// TIA Portal V18 export
FUNCTION "SS1_A1_CPU1215_IO_Update" : Void   // FC11010, LAD
{ S7_Optimized_Access := 'TRUE' }
VERSION : 0.1
// stored: AutoNumber false, IsIECCheckEnabled false, SetENOAutomatically false, UDAEnableTagReadback false
BEGIN

REGION Network 1: AI0 / "AI01.1.1" iw64
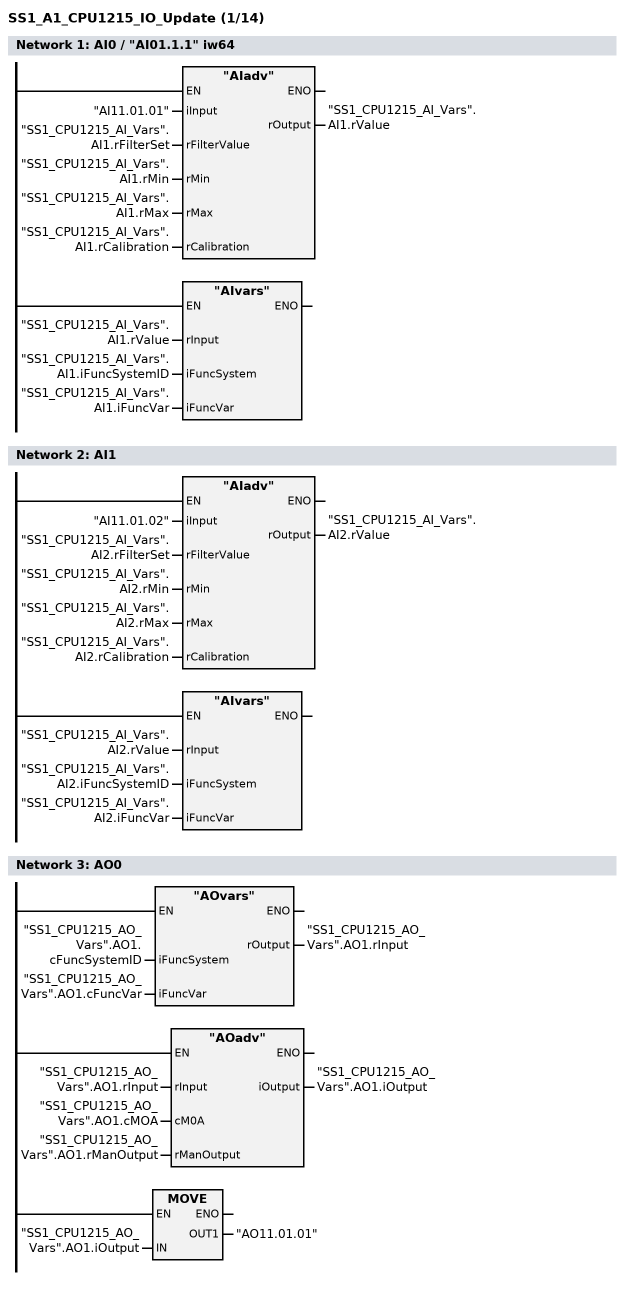
   RUNG wire#powerrail
      "AIadv"(iInput := "AI11.01.01", rFilterValue := "SS1_CPU1215_AI_Vars".AI1.rFilterSet, rMin := "SS1_CPU1215_AI_Vars".AI1.rMin, rMax := "SS1_CPU1215_AI_Vars".AI1.rMax, rCalibration := "SS1_CPU1215_AI_Vars".AI1.rCalibration, rOutput => "SS1_CPU1215_AI_Vars".AI1.rValue)
   END_RUNG
   RUNG wire#powerrail
      "AIvars"(rInput := "SS1_CPU1215_AI_Vars".AI1.rValue, iFuncSystem := "SS1_CPU1215_AI_Vars".AI1.iFuncSystemID, iFuncVar := "SS1_CPU1215_AI_Vars".AI1.iFuncVar)
   END_RUNG
   // the same network as SCL:
   "AIadv"(iInput := "AI11.01.01",
           rFilterValue := "SS1_CPU1215_AI_Vars".AI1.rFilterSet,
           rMin := "SS1_CPU1215_AI_Vars".AI1.rMin,
           rMax := "SS1_CPU1215_AI_Vars".AI1.rMax,
           rCalibration := "SS1_CPU1215_AI_Vars".AI1.rCalibration,
           rOutput => "SS1_CPU1215_AI_Vars".AI1.rValue);
   "AIvars"(rInput := "SS1_CPU1215_AI_Vars".AI1.rValue,
            iFuncSystem := "SS1_CPU1215_AI_Vars".AI1.iFuncSystemID,
            iFuncVar := "SS1_CPU1215_AI_Vars".AI1.iFuncVar);
END_REGION

REGION Network 2: AI1
   RUNG wire#powerrail
      "AIadv"(iInput := "AI11.01.02", rFilterValue := "SS1_CPU1215_AI_Vars".AI2.rFilterSet, rMin := "SS1_CPU1215_AI_Vars".AI2.rMin, rMax := "SS1_CPU1215_AI_Vars".AI2.rMax, rCalibration := "SS1_CPU1215_AI_Vars".AI2.rCalibration, rOutput => "SS1_CPU1215_AI_Vars".AI2.rValue)
   END_RUNG
   RUNG wire#powerrail
      "AIvars"(rInput := "SS1_CPU1215_AI_Vars".AI2.rValue, iFuncSystem := "SS1_CPU1215_AI_Vars".AI2.iFuncSystemID, iFuncVar := "SS1_CPU1215_AI_Vars".AI2.iFuncVar)
   END_RUNG
   // the same network as SCL:
   "AIadv"(iInput := "AI11.01.02",
           rFilterValue := "SS1_CPU1215_AI_Vars".AI2.rFilterSet,
           rMin := "SS1_CPU1215_AI_Vars".AI2.rMin,
           rMax := "SS1_CPU1215_AI_Vars".AI2.rMax,
           rCalibration := "SS1_CPU1215_AI_Vars".AI2.rCalibration,
           rOutput => "SS1_CPU1215_AI_Vars".AI2.rValue);
   "AIvars"(rInput := "SS1_CPU1215_AI_Vars".AI2.rValue,
            iFuncSystem := "SS1_CPU1215_AI_Vars".AI2.iFuncSystemID,
            iFuncVar := "SS1_CPU1215_AI_Vars".AI2.iFuncVar);
END_REGION

REGION Network 3: AO0
   RUNG wire#powerrail
      "AOvars"(iFuncSystem := "SS1_CPU1215_AO_Vars".AO1.cFuncSystemID, iFuncVar := "SS1_CPU1215_AO_Vars".AO1.cFuncVar, rOutput => "SS1_CPU1215_AO_Vars".AO1.rInput)
   END_RUNG
   RUNG wire#powerrail
      "AOadv"(rInput := "SS1_CPU1215_AO_Vars".AO1.rInput, cM0A := "SS1_CPU1215_AO_Vars".AO1.cMOA, rManOutput := "SS1_CPU1215_AO_Vars".AO1.rManOutput, iOutput => "SS1_CPU1215_AO_Vars".AO1.iOutput)
   END_RUNG
   RUNG wire#powerrail
      Move(in := "SS1_CPU1215_AO_Vars".AO1.iOutput, out1 => "AO11.01.01")
   END_RUNG
   // the same network as SCL:
   "AOvars"(iFuncSystem := "SS1_CPU1215_AO_Vars".AO1.cFuncSystemID,
            iFuncVar := "SS1_CPU1215_AO_Vars".AO1.cFuncVar,
            rOutput => "SS1_CPU1215_AO_Vars".AO1.rInput);
   "AOadv"(rInput := "SS1_CPU1215_AO_Vars".AO1.rInput,
           cM0A := "SS1_CPU1215_AO_Vars".AO1.cMOA,
           rManOutput := "SS1_CPU1215_AO_Vars".AO1.rManOutput,
           iOutput => "SS1_CPU1215_AO_Vars".AO1.iOutput);
   "AO11.01.01" := "SS1_CPU1215_AO_Vars".AO1.iOutput;
END_REGION

REGION Network 4: AO1
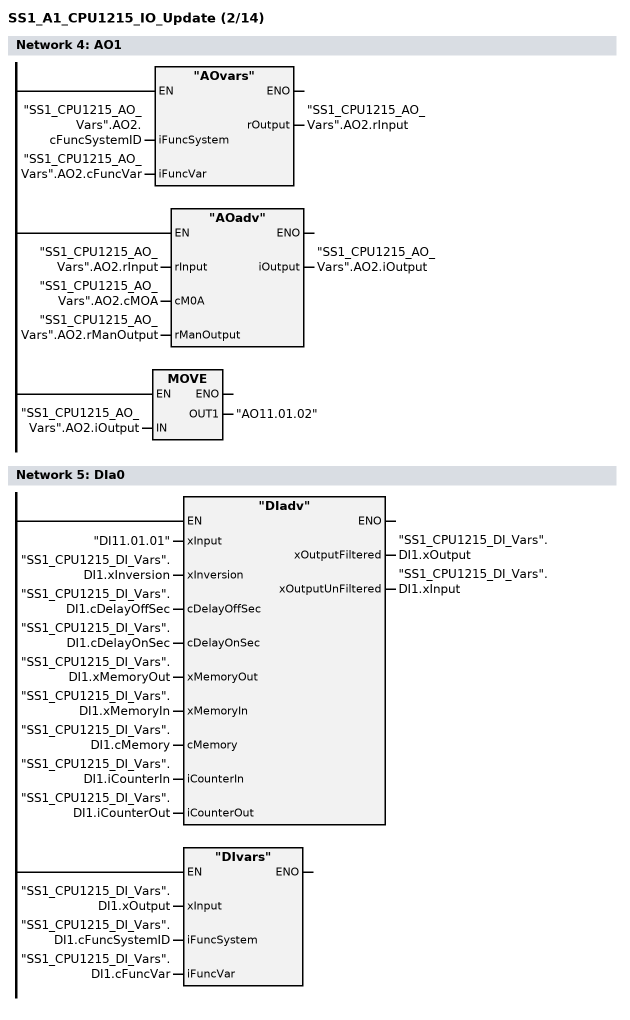
   RUNG wire#powerrail
      "AOvars"(iFuncSystem := "SS1_CPU1215_AO_Vars".AO2.cFuncSystemID, iFuncVar := "SS1_CPU1215_AO_Vars".AO2.cFuncVar, rOutput => "SS1_CPU1215_AO_Vars".AO2.rInput)
   END_RUNG
   RUNG wire#powerrail
      "AOadv"(rInput := "SS1_CPU1215_AO_Vars".AO2.rInput, cM0A := "SS1_CPU1215_AO_Vars".AO2.cMOA, rManOutput := "SS1_CPU1215_AO_Vars".AO2.rManOutput, iOutput => "SS1_CPU1215_AO_Vars".AO2.iOutput)
   END_RUNG
   RUNG wire#powerrail
      Move(in := "SS1_CPU1215_AO_Vars".AO2.iOutput, out1 => "AO11.01.02")
   END_RUNG
   // the same network as SCL:
   "AOvars"(iFuncSystem := "SS1_CPU1215_AO_Vars".AO2.cFuncSystemID,
            iFuncVar := "SS1_CPU1215_AO_Vars".AO2.cFuncVar,
            rOutput => "SS1_CPU1215_AO_Vars".AO2.rInput);
   "AOadv"(rInput := "SS1_CPU1215_AO_Vars".AO2.rInput,
           cM0A := "SS1_CPU1215_AO_Vars".AO2.cMOA,
           rManOutput := "SS1_CPU1215_AO_Vars".AO2.rManOutput,
           iOutput => "SS1_CPU1215_AO_Vars".AO2.iOutput);
   "AO11.01.02" := "SS1_CPU1215_AO_Vars".AO2.iOutput;
END_REGION

REGION Network 5: DIa0
   RUNG wire#powerrail
      "DIadv"(xInput := "DI11.01.01", xInversion := "SS1_CPU1215_DI_Vars".DI1.xInversion, cDelayOffSec := "SS1_CPU1215_DI_Vars".DI1.cDelayOffSec, cDelayOnSec := "SS1_CPU1215_DI_Vars".DI1.cDelayOnSec, xMemoryOut := "SS1_CPU1215_DI_Vars".DI1.xMemoryOut, xMemoryIn := "SS1_CPU1215_DI_Vars".DI1.xMemoryIn, cMemory := "SS1_CPU1215_DI_Vars".DI1.cMemory, xOutputFiltered => "SS1_CPU1215_DI_Vars".DI1.xOutput, xOutputUnFiltered => "SS1_CPU1215_DI_Vars".DI1.xInput, iCounterIn := "SS1_CPU1215_DI_Vars".DI1.iCounterIn, iCounterOut := "SS1_CPU1215_DI_Vars".DI1.iCounterOut)
   END_RUNG
   RUNG wire#powerrail
      "DIvars"(xInput := "SS1_CPU1215_DI_Vars".DI1.xOutput, iFuncSystem := "SS1_CPU1215_DI_Vars".DI1.cFuncSystemID, iFuncVar := "SS1_CPU1215_DI_Vars".DI1.cFuncVar)
   END_RUNG
   // the same network as SCL:
   "DIadv"(xInput := "DI11.01.01",
           xInversion := "SS1_CPU1215_DI_Vars".DI1.xInversion,
           cDelayOffSec := "SS1_CPU1215_DI_Vars".DI1.cDelayOffSec,
           cDelayOnSec := "SS1_CPU1215_DI_Vars".DI1.cDelayOnSec,
           xMemoryOut := "SS1_CPU1215_DI_Vars".DI1.xMemoryOut,
           xMemoryIn := "SS1_CPU1215_DI_Vars".DI1.xMemoryIn,
           cMemory := "SS1_CPU1215_DI_Vars".DI1.cMemory,
           iCounterIn := "SS1_CPU1215_DI_Vars".DI1.iCounterIn,
           iCounterOut := "SS1_CPU1215_DI_Vars".DI1.iCounterOut,
           xOutputFiltered => "SS1_CPU1215_DI_Vars".DI1.xOutput,
           xOutputUnFiltered => "SS1_CPU1215_DI_Vars".DI1.xInput);
   "DIvars"(xInput := "SS1_CPU1215_DI_Vars".DI1.xOutput,
            iFuncSystem := "SS1_CPU1215_DI_Vars".DI1.cFuncSystemID,
            iFuncVar := "SS1_CPU1215_DI_Vars".DI1.cFuncVar);
END_REGION

REGION Network 6: DIa1
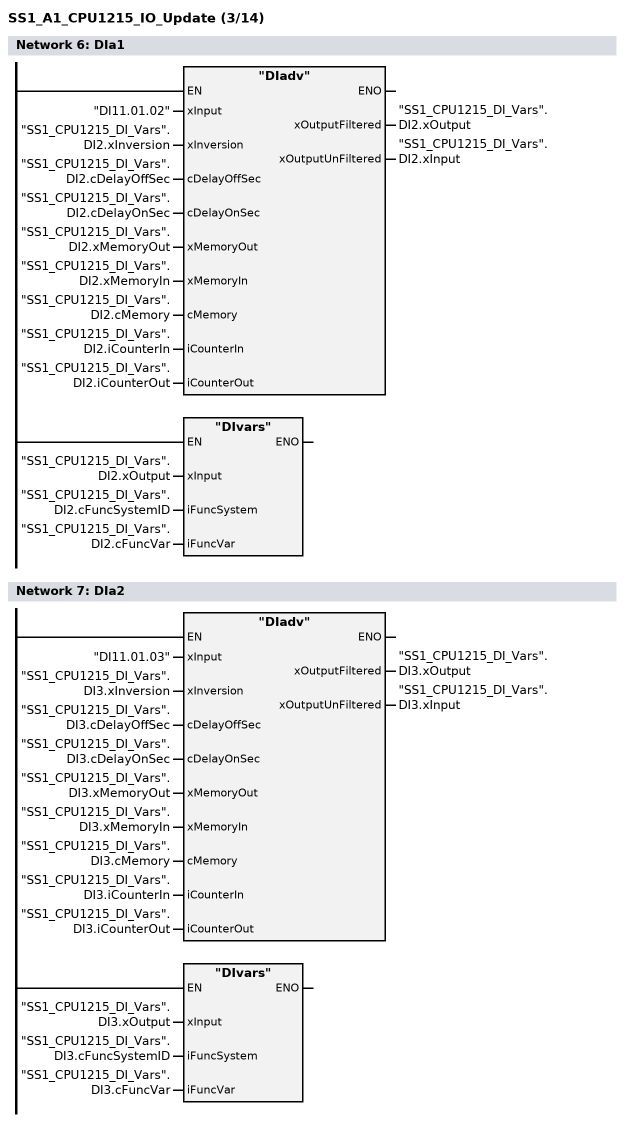
   RUNG wire#powerrail
      "DIadv"(xInput := "DI11.01.02", xInversion := "SS1_CPU1215_DI_Vars".DI2.xInversion, cDelayOffSec := "SS1_CPU1215_DI_Vars".DI2.cDelayOffSec, cDelayOnSec := "SS1_CPU1215_DI_Vars".DI2.cDelayOnSec, xMemoryOut := "SS1_CPU1215_DI_Vars".DI2.xMemoryOut, xMemoryIn := "SS1_CPU1215_DI_Vars".DI2.xMemoryIn, cMemory := "SS1_CPU1215_DI_Vars".DI2.cMemory, xOutputFiltered => "SS1_CPU1215_DI_Vars".DI2.xOutput, xOutputUnFiltered => "SS1_CPU1215_DI_Vars".DI2.xInput, iCounterIn := "SS1_CPU1215_DI_Vars".DI2.iCounterIn, iCounterOut := "SS1_CPU1215_DI_Vars".DI2.iCounterOut)
   END_RUNG
   RUNG wire#powerrail
      "DIvars"(xInput := "SS1_CPU1215_DI_Vars".DI2.xOutput, iFuncSystem := "SS1_CPU1215_DI_Vars".DI2.cFuncSystemID, iFuncVar := "SS1_CPU1215_DI_Vars".DI2.cFuncVar)
   END_RUNG
   // the same network as SCL:
   "DIadv"(xInput := "DI11.01.02",
           xInversion := "SS1_CPU1215_DI_Vars".DI2.xInversion,
           cDelayOffSec := "SS1_CPU1215_DI_Vars".DI2.cDelayOffSec,
           cDelayOnSec := "SS1_CPU1215_DI_Vars".DI2.cDelayOnSec,
           xMemoryOut := "SS1_CPU1215_DI_Vars".DI2.xMemoryOut,
           xMemoryIn := "SS1_CPU1215_DI_Vars".DI2.xMemoryIn,
           cMemory := "SS1_CPU1215_DI_Vars".DI2.cMemory,
           iCounterIn := "SS1_CPU1215_DI_Vars".DI2.iCounterIn,
           iCounterOut := "SS1_CPU1215_DI_Vars".DI2.iCounterOut,
           xOutputFiltered => "SS1_CPU1215_DI_Vars".DI2.xOutput,
           xOutputUnFiltered => "SS1_CPU1215_DI_Vars".DI2.xInput);
   "DIvars"(xInput := "SS1_CPU1215_DI_Vars".DI2.xOutput,
            iFuncSystem := "SS1_CPU1215_DI_Vars".DI2.cFuncSystemID,
            iFuncVar := "SS1_CPU1215_DI_Vars".DI2.cFuncVar);
END_REGION

REGION Network 7: DIa2
   RUNG wire#powerrail
      "DIadv"(xInput := "DI11.01.03", xInversion := "SS1_CPU1215_DI_Vars".DI3.xInversion, cDelayOffSec := "SS1_CPU1215_DI_Vars".DI3.cDelayOffSec, cDelayOnSec := "SS1_CPU1215_DI_Vars".DI3.cDelayOnSec, xMemoryOut := "SS1_CPU1215_DI_Vars".DI3.xMemoryOut, xMemoryIn := "SS1_CPU1215_DI_Vars".DI3.xMemoryIn, cMemory := "SS1_CPU1215_DI_Vars".DI3.cMemory, xOutputFiltered => "SS1_CPU1215_DI_Vars".DI3.xOutput, xOutputUnFiltered => "SS1_CPU1215_DI_Vars".DI3.xInput, iCounterIn := "SS1_CPU1215_DI_Vars".DI3.iCounterIn, iCounterOut := "SS1_CPU1215_DI_Vars".DI3.iCounterOut)
   END_RUNG
   RUNG wire#powerrail
      "DIvars"(xInput := "SS1_CPU1215_DI_Vars".DI3.xOutput, iFuncSystem := "SS1_CPU1215_DI_Vars".DI3.cFuncSystemID, iFuncVar := "SS1_CPU1215_DI_Vars".DI3.cFuncVar)
   END_RUNG
   // the same network as SCL:
   "DIadv"(xInput := "DI11.01.03",
           xInversion := "SS1_CPU1215_DI_Vars".DI3.xInversion,
           cDelayOffSec := "SS1_CPU1215_DI_Vars".DI3.cDelayOffSec,
           cDelayOnSec := "SS1_CPU1215_DI_Vars".DI3.cDelayOnSec,
           xMemoryOut := "SS1_CPU1215_DI_Vars".DI3.xMemoryOut,
           xMemoryIn := "SS1_CPU1215_DI_Vars".DI3.xMemoryIn,
           cMemory := "SS1_CPU1215_DI_Vars".DI3.cMemory,
           iCounterIn := "SS1_CPU1215_DI_Vars".DI3.iCounterIn,
           iCounterOut := "SS1_CPU1215_DI_Vars".DI3.iCounterOut,
           xOutputFiltered => "SS1_CPU1215_DI_Vars".DI3.xOutput,
           xOutputUnFiltered => "SS1_CPU1215_DI_Vars".DI3.xInput);
   "DIvars"(xInput := "SS1_CPU1215_DI_Vars".DI3.xOutput,
            iFuncSystem := "SS1_CPU1215_DI_Vars".DI3.cFuncSystemID,
            iFuncVar := "SS1_CPU1215_DI_Vars".DI3.cFuncVar);
END_REGION

REGION Network 8: DIa3
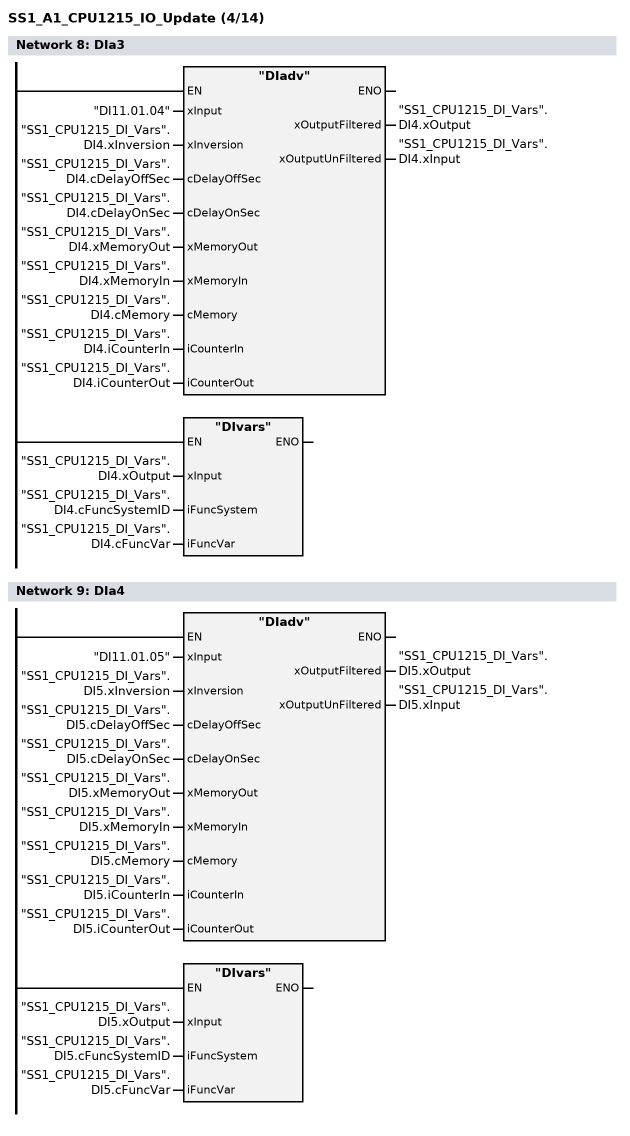
   RUNG wire#powerrail
      "DIadv"(xInput := "DI11.01.04", xInversion := "SS1_CPU1215_DI_Vars".DI4.xInversion, cDelayOffSec := "SS1_CPU1215_DI_Vars".DI4.cDelayOffSec, cDelayOnSec := "SS1_CPU1215_DI_Vars".DI4.cDelayOnSec, xMemoryOut := "SS1_CPU1215_DI_Vars".DI4.xMemoryOut, xMemoryIn := "SS1_CPU1215_DI_Vars".DI4.xMemoryIn, cMemory := "SS1_CPU1215_DI_Vars".DI4.cMemory, xOutputFiltered => "SS1_CPU1215_DI_Vars".DI4.xOutput, xOutputUnFiltered => "SS1_CPU1215_DI_Vars".DI4.xInput, iCounterIn := "SS1_CPU1215_DI_Vars".DI4.iCounterIn, iCounterOut := "SS1_CPU1215_DI_Vars".DI4.iCounterOut)
   END_RUNG
   RUNG wire#powerrail
      "DIvars"(xInput := "SS1_CPU1215_DI_Vars".DI4.xOutput, iFuncSystem := "SS1_CPU1215_DI_Vars".DI4.cFuncSystemID, iFuncVar := "SS1_CPU1215_DI_Vars".DI4.cFuncVar)
   END_RUNG
   // the same network as SCL:
   "DIadv"(xInput := "DI11.01.04",
           xInversion := "SS1_CPU1215_DI_Vars".DI4.xInversion,
           cDelayOffSec := "SS1_CPU1215_DI_Vars".DI4.cDelayOffSec,
           cDelayOnSec := "SS1_CPU1215_DI_Vars".DI4.cDelayOnSec,
           xMemoryOut := "SS1_CPU1215_DI_Vars".DI4.xMemoryOut,
           xMemoryIn := "SS1_CPU1215_DI_Vars".DI4.xMemoryIn,
           cMemory := "SS1_CPU1215_DI_Vars".DI4.cMemory,
           iCounterIn := "SS1_CPU1215_DI_Vars".DI4.iCounterIn,
           iCounterOut := "SS1_CPU1215_DI_Vars".DI4.iCounterOut,
           xOutputFiltered => "SS1_CPU1215_DI_Vars".DI4.xOutput,
           xOutputUnFiltered => "SS1_CPU1215_DI_Vars".DI4.xInput);
   "DIvars"(xInput := "SS1_CPU1215_DI_Vars".DI4.xOutput,
            iFuncSystem := "SS1_CPU1215_DI_Vars".DI4.cFuncSystemID,
            iFuncVar := "SS1_CPU1215_DI_Vars".DI4.cFuncVar);
END_REGION

REGION Network 9: DIa4
   RUNG wire#powerrail
      "DIadv"(xInput := "DI11.01.05", xInversion := "SS1_CPU1215_DI_Vars".DI5.xInversion, cDelayOffSec := "SS1_CPU1215_DI_Vars".DI5.cDelayOffSec, cDelayOnSec := "SS1_CPU1215_DI_Vars".DI5.cDelayOnSec, xMemoryOut := "SS1_CPU1215_DI_Vars".DI5.xMemoryOut, xMemoryIn := "SS1_CPU1215_DI_Vars".DI5.xMemoryIn, cMemory := "SS1_CPU1215_DI_Vars".DI5.cMemory, xOutputFiltered => "SS1_CPU1215_DI_Vars".DI5.xOutput, xOutputUnFiltered => "SS1_CPU1215_DI_Vars".DI5.xInput, iCounterIn := "SS1_CPU1215_DI_Vars".DI5.iCounterIn, iCounterOut := "SS1_CPU1215_DI_Vars".DI5.iCounterOut)
   END_RUNG
   RUNG wire#powerrail
      "DIvars"(xInput := "SS1_CPU1215_DI_Vars".DI5.xOutput, iFuncSystem := "SS1_CPU1215_DI_Vars".DI5.cFuncSystemID, iFuncVar := "SS1_CPU1215_DI_Vars".DI5.cFuncVar)
   END_RUNG
   // the same network as SCL:
   "DIadv"(xInput := "DI11.01.05",
           xInversion := "SS1_CPU1215_DI_Vars".DI5.xInversion,
           cDelayOffSec := "SS1_CPU1215_DI_Vars".DI5.cDelayOffSec,
           cDelayOnSec := "SS1_CPU1215_DI_Vars".DI5.cDelayOnSec,
           xMemoryOut := "SS1_CPU1215_DI_Vars".DI5.xMemoryOut,
           xMemoryIn := "SS1_CPU1215_DI_Vars".DI5.xMemoryIn,
           cMemory := "SS1_CPU1215_DI_Vars".DI5.cMemory,
           iCounterIn := "SS1_CPU1215_DI_Vars".DI5.iCounterIn,
           iCounterOut := "SS1_CPU1215_DI_Vars".DI5.iCounterOut,
           xOutputFiltered => "SS1_CPU1215_DI_Vars".DI5.xOutput,
           xOutputUnFiltered => "SS1_CPU1215_DI_Vars".DI5.xInput);
   "DIvars"(xInput := "SS1_CPU1215_DI_Vars".DI5.xOutput,
            iFuncSystem := "SS1_CPU1215_DI_Vars".DI5.cFuncSystemID,
            iFuncVar := "SS1_CPU1215_DI_Vars".DI5.cFuncVar);
END_REGION

REGION Network 10: DIa5
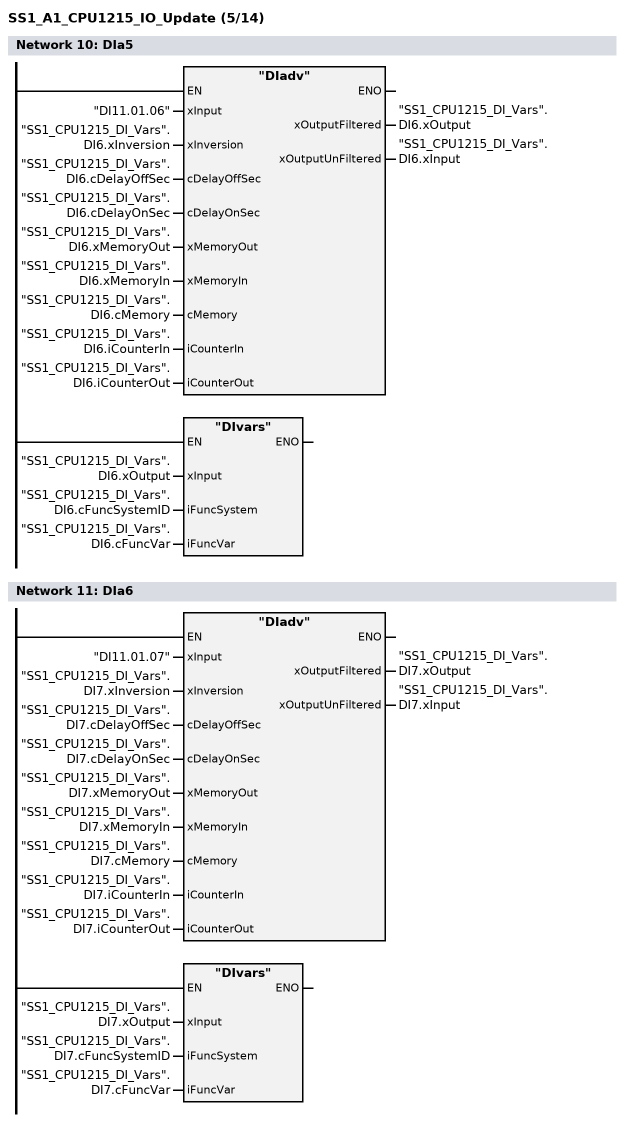
   RUNG wire#powerrail
      "DIadv"(xInput := "DI11.01.06", xInversion := "SS1_CPU1215_DI_Vars".DI6.xInversion, cDelayOffSec := "SS1_CPU1215_DI_Vars".DI6.cDelayOffSec, cDelayOnSec := "SS1_CPU1215_DI_Vars".DI6.cDelayOnSec, xMemoryOut := "SS1_CPU1215_DI_Vars".DI6.xMemoryOut, xMemoryIn := "SS1_CPU1215_DI_Vars".DI6.xMemoryIn, cMemory := "SS1_CPU1215_DI_Vars".DI6.cMemory, xOutputFiltered => "SS1_CPU1215_DI_Vars".DI6.xOutput, xOutputUnFiltered => "SS1_CPU1215_DI_Vars".DI6.xInput, iCounterIn := "SS1_CPU1215_DI_Vars".DI6.iCounterIn, iCounterOut := "SS1_CPU1215_DI_Vars".DI6.iCounterOut)
   END_RUNG
   RUNG wire#powerrail
      "DIvars"(xInput := "SS1_CPU1215_DI_Vars".DI6.xOutput, iFuncSystem := "SS1_CPU1215_DI_Vars".DI6.cFuncSystemID, iFuncVar := "SS1_CPU1215_DI_Vars".DI6.cFuncVar)
   END_RUNG
   // the same network as SCL:
   "DIadv"(xInput := "DI11.01.06",
           xInversion := "SS1_CPU1215_DI_Vars".DI6.xInversion,
           cDelayOffSec := "SS1_CPU1215_DI_Vars".DI6.cDelayOffSec,
           cDelayOnSec := "SS1_CPU1215_DI_Vars".DI6.cDelayOnSec,
           xMemoryOut := "SS1_CPU1215_DI_Vars".DI6.xMemoryOut,
           xMemoryIn := "SS1_CPU1215_DI_Vars".DI6.xMemoryIn,
           cMemory := "SS1_CPU1215_DI_Vars".DI6.cMemory,
           iCounterIn := "SS1_CPU1215_DI_Vars".DI6.iCounterIn,
           iCounterOut := "SS1_CPU1215_DI_Vars".DI6.iCounterOut,
           xOutputFiltered => "SS1_CPU1215_DI_Vars".DI6.xOutput,
           xOutputUnFiltered => "SS1_CPU1215_DI_Vars".DI6.xInput);
   "DIvars"(xInput := "SS1_CPU1215_DI_Vars".DI6.xOutput,
            iFuncSystem := "SS1_CPU1215_DI_Vars".DI6.cFuncSystemID,
            iFuncVar := "SS1_CPU1215_DI_Vars".DI6.cFuncVar);
END_REGION

REGION Network 11: DIa6
   RUNG wire#powerrail
      "DIadv"(xInput := "DI11.01.07", xInversion := "SS1_CPU1215_DI_Vars".DI7.xInversion, cDelayOffSec := "SS1_CPU1215_DI_Vars".DI7.cDelayOffSec, cDelayOnSec := "SS1_CPU1215_DI_Vars".DI7.cDelayOnSec, xMemoryOut := "SS1_CPU1215_DI_Vars".DI7.xMemoryOut, xMemoryIn := "SS1_CPU1215_DI_Vars".DI7.xMemoryIn, cMemory := "SS1_CPU1215_DI_Vars".DI7.cMemory, xOutputFiltered => "SS1_CPU1215_DI_Vars".DI7.xOutput, xOutputUnFiltered => "SS1_CPU1215_DI_Vars".DI7.xInput, iCounterIn := "SS1_CPU1215_DI_Vars".DI7.iCounterIn, iCounterOut := "SS1_CPU1215_DI_Vars".DI7.iCounterOut)
   END_RUNG
   RUNG wire#powerrail
      "DIvars"(xInput := "SS1_CPU1215_DI_Vars".DI7.xOutput, iFuncSystem := "SS1_CPU1215_DI_Vars".DI7.cFuncSystemID, iFuncVar := "SS1_CPU1215_DI_Vars".DI7.cFuncVar)
   END_RUNG
   // the same network as SCL:
   "DIadv"(xInput := "DI11.01.07",
           xInversion := "SS1_CPU1215_DI_Vars".DI7.xInversion,
           cDelayOffSec := "SS1_CPU1215_DI_Vars".DI7.cDelayOffSec,
           cDelayOnSec := "SS1_CPU1215_DI_Vars".DI7.cDelayOnSec,
           xMemoryOut := "SS1_CPU1215_DI_Vars".DI7.xMemoryOut,
           xMemoryIn := "SS1_CPU1215_DI_Vars".DI7.xMemoryIn,
           cMemory := "SS1_CPU1215_DI_Vars".DI7.cMemory,
           iCounterIn := "SS1_CPU1215_DI_Vars".DI7.iCounterIn,
           iCounterOut := "SS1_CPU1215_DI_Vars".DI7.iCounterOut,
           xOutputFiltered => "SS1_CPU1215_DI_Vars".DI7.xOutput,
           xOutputUnFiltered => "SS1_CPU1215_DI_Vars".DI7.xInput);
   "DIvars"(xInput := "SS1_CPU1215_DI_Vars".DI7.xOutput,
            iFuncSystem := "SS1_CPU1215_DI_Vars".DI7.cFuncSystemID,
            iFuncVar := "SS1_CPU1215_DI_Vars".DI7.cFuncVar);
END_REGION

REGION Network 12: DIa7 / DI01.1.08 EDP під охороною
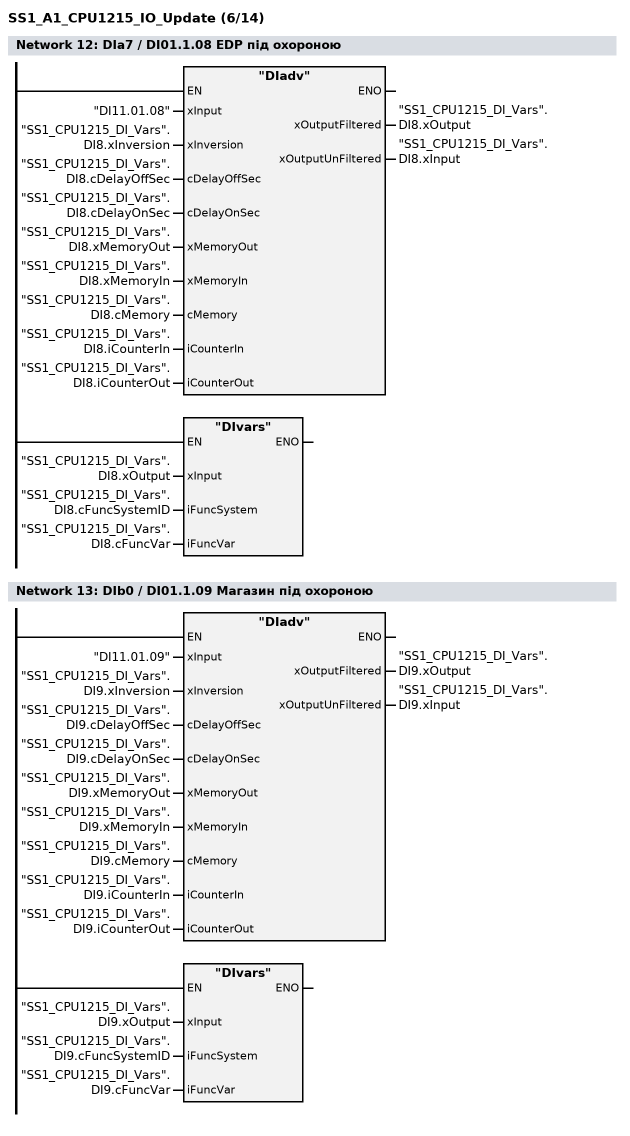
   RUNG wire#powerrail
      "DIadv"(xInput := "DI11.01.08", xInversion := "SS1_CPU1215_DI_Vars".DI8.xInversion, cDelayOffSec := "SS1_CPU1215_DI_Vars".DI8.cDelayOffSec, cDelayOnSec := "SS1_CPU1215_DI_Vars".DI8.cDelayOnSec, xMemoryOut := "SS1_CPU1215_DI_Vars".DI8.xMemoryOut, xMemoryIn := "SS1_CPU1215_DI_Vars".DI8.xMemoryIn, cMemory := "SS1_CPU1215_DI_Vars".DI8.cMemory, iCounterIn := "SS1_CPU1215_DI_Vars".DI8.iCounterIn, iCounterOut := "SS1_CPU1215_DI_Vars".DI8.iCounterOut, xOutputFiltered => "SS1_CPU1215_DI_Vars".DI8.xOutput, xOutputUnFiltered => "SS1_CPU1215_DI_Vars".DI8.xInput)
   END_RUNG
   RUNG wire#powerrail
      "DIvars"(xInput := "SS1_CPU1215_DI_Vars".DI8.xOutput, iFuncSystem := "SS1_CPU1215_DI_Vars".DI8.cFuncSystemID, iFuncVar := "SS1_CPU1215_DI_Vars".DI8.cFuncVar)
   END_RUNG
   // the same network as SCL:
   "DIadv"(xInput := "DI11.01.08",
           xInversion := "SS1_CPU1215_DI_Vars".DI8.xInversion,
           cDelayOffSec := "SS1_CPU1215_DI_Vars".DI8.cDelayOffSec,
           cDelayOnSec := "SS1_CPU1215_DI_Vars".DI8.cDelayOnSec,
           xMemoryOut := "SS1_CPU1215_DI_Vars".DI8.xMemoryOut,
           xMemoryIn := "SS1_CPU1215_DI_Vars".DI8.xMemoryIn,
           cMemory := "SS1_CPU1215_DI_Vars".DI8.cMemory,
           iCounterIn := "SS1_CPU1215_DI_Vars".DI8.iCounterIn,
           iCounterOut := "SS1_CPU1215_DI_Vars".DI8.iCounterOut,
           xOutputFiltered => "SS1_CPU1215_DI_Vars".DI8.xOutput,
           xOutputUnFiltered => "SS1_CPU1215_DI_Vars".DI8.xInput);
   "DIvars"(xInput := "SS1_CPU1215_DI_Vars".DI8.xOutput,
            iFuncSystem := "SS1_CPU1215_DI_Vars".DI8.cFuncSystemID,
            iFuncVar := "SS1_CPU1215_DI_Vars".DI8.cFuncVar);
END_REGION

REGION Network 13: DIb0 / DI01.1.09 Магазин під охороною
   RUNG wire#powerrail
      "DIadv"(xInput := "DI11.01.09", xInversion := "SS1_CPU1215_DI_Vars".DI9.xInversion, cDelayOffSec := "SS1_CPU1215_DI_Vars".DI9.cDelayOffSec, cDelayOnSec := "SS1_CPU1215_DI_Vars".DI9.cDelayOnSec, xMemoryOut := "SS1_CPU1215_DI_Vars".DI9.xMemoryOut, xMemoryIn := "SS1_CPU1215_DI_Vars".DI9.xMemoryIn, cMemory := "SS1_CPU1215_DI_Vars".DI9.cMemory, xOutputFiltered => "SS1_CPU1215_DI_Vars".DI9.xOutput, xOutputUnFiltered => "SS1_CPU1215_DI_Vars".DI9.xInput, iCounterIn := "SS1_CPU1215_DI_Vars".DI9.iCounterIn, iCounterOut := "SS1_CPU1215_DI_Vars".DI9.iCounterOut)
   END_RUNG
   RUNG wire#powerrail
      "DIvars"(xInput := "SS1_CPU1215_DI_Vars".DI9.xOutput, iFuncSystem := "SS1_CPU1215_DI_Vars".DI9.cFuncSystemID, iFuncVar := "SS1_CPU1215_DI_Vars".DI9.cFuncVar)
   END_RUNG
   // the same network as SCL:
   "DIadv"(xInput := "DI11.01.09",
           xInversion := "SS1_CPU1215_DI_Vars".DI9.xInversion,
           cDelayOffSec := "SS1_CPU1215_DI_Vars".DI9.cDelayOffSec,
           cDelayOnSec := "SS1_CPU1215_DI_Vars".DI9.cDelayOnSec,
           xMemoryOut := "SS1_CPU1215_DI_Vars".DI9.xMemoryOut,
           xMemoryIn := "SS1_CPU1215_DI_Vars".DI9.xMemoryIn,
           cMemory := "SS1_CPU1215_DI_Vars".DI9.cMemory,
           iCounterIn := "SS1_CPU1215_DI_Vars".DI9.iCounterIn,
           iCounterOut := "SS1_CPU1215_DI_Vars".DI9.iCounterOut,
           xOutputFiltered => "SS1_CPU1215_DI_Vars".DI9.xOutput,
           xOutputUnFiltered => "SS1_CPU1215_DI_Vars".DI9.xInput);
   "DIvars"(xInput := "SS1_CPU1215_DI_Vars".DI9.xOutput,
            iFuncSystem := "SS1_CPU1215_DI_Vars".DI9.cFuncSystemID,
            iFuncVar := "SS1_CPU1215_DI_Vars".DI9.cFuncVar);
END_REGION

REGION Network 14: DIb1 / DI01.1.10 Аварійний рівень загазованості
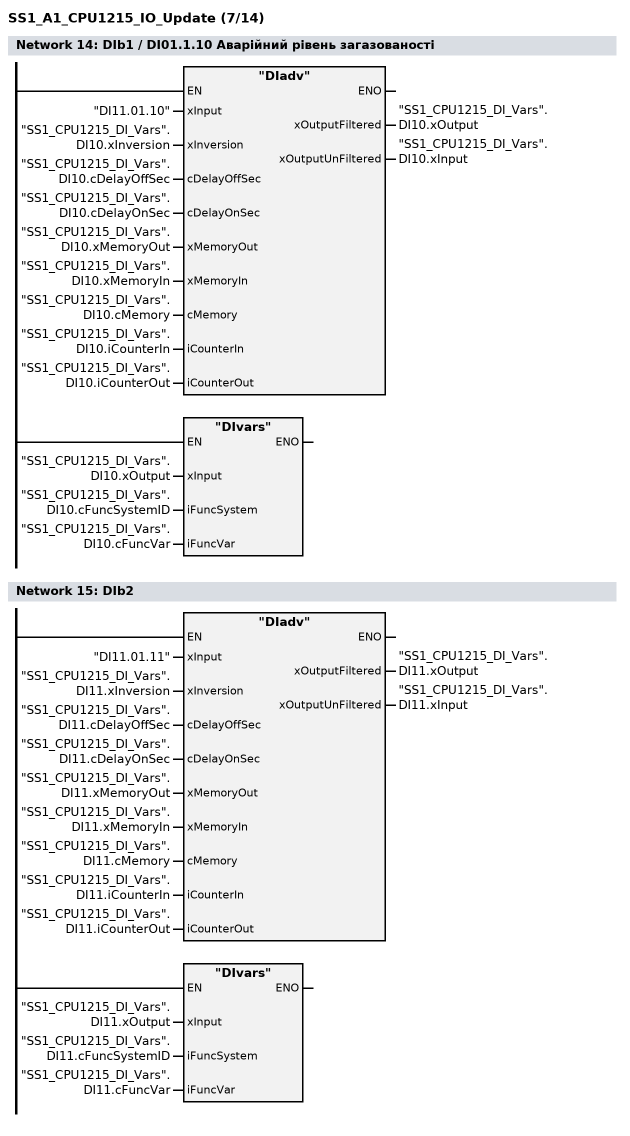
   RUNG wire#powerrail
      "DIadv"(xInput := "DI11.01.10", xInversion := "SS1_CPU1215_DI_Vars".DI10.xInversion, cDelayOffSec := "SS1_CPU1215_DI_Vars".DI10.cDelayOffSec, cDelayOnSec := "SS1_CPU1215_DI_Vars".DI10.cDelayOnSec, xMemoryOut := "SS1_CPU1215_DI_Vars".DI10.xMemoryOut, xMemoryIn := "SS1_CPU1215_DI_Vars".DI10.xMemoryIn, cMemory := "SS1_CPU1215_DI_Vars".DI10.cMemory, xOutputFiltered => "SS1_CPU1215_DI_Vars".DI10.xOutput, xOutputUnFiltered => "SS1_CPU1215_DI_Vars".DI10.xInput, iCounterIn := "SS1_CPU1215_DI_Vars".DI10.iCounterIn, iCounterOut := "SS1_CPU1215_DI_Vars".DI10.iCounterOut)
   END_RUNG
   RUNG wire#powerrail
      "DIvars"(xInput := "SS1_CPU1215_DI_Vars".DI10.xOutput, iFuncSystem := "SS1_CPU1215_DI_Vars".DI10.cFuncSystemID, iFuncVar := "SS1_CPU1215_DI_Vars".DI10.cFuncVar)
   END_RUNG
   // the same network as SCL:
   "DIadv"(xInput := "DI11.01.10",
           xInversion := "SS1_CPU1215_DI_Vars".DI10.xInversion,
           cDelayOffSec := "SS1_CPU1215_DI_Vars".DI10.cDelayOffSec,
           cDelayOnSec := "SS1_CPU1215_DI_Vars".DI10.cDelayOnSec,
           xMemoryOut := "SS1_CPU1215_DI_Vars".DI10.xMemoryOut,
           xMemoryIn := "SS1_CPU1215_DI_Vars".DI10.xMemoryIn,
           cMemory := "SS1_CPU1215_DI_Vars".DI10.cMemory,
           iCounterIn := "SS1_CPU1215_DI_Vars".DI10.iCounterIn,
           iCounterOut := "SS1_CPU1215_DI_Vars".DI10.iCounterOut,
           xOutputFiltered => "SS1_CPU1215_DI_Vars".DI10.xOutput,
           xOutputUnFiltered => "SS1_CPU1215_DI_Vars".DI10.xInput);
   "DIvars"(xInput := "SS1_CPU1215_DI_Vars".DI10.xOutput,
            iFuncSystem := "SS1_CPU1215_DI_Vars".DI10.cFuncSystemID,
            iFuncVar := "SS1_CPU1215_DI_Vars".DI10.cFuncVar);
END_REGION

REGION Network 15: DIb2
   RUNG wire#powerrail
      "DIadv"(xInput := "DI11.01.11", xInversion := "SS1_CPU1215_DI_Vars".DI11.xInversion, cDelayOffSec := "SS1_CPU1215_DI_Vars".DI11.cDelayOffSec, cDelayOnSec := "SS1_CPU1215_DI_Vars".DI11.cDelayOnSec, xMemoryOut := "SS1_CPU1215_DI_Vars".DI11.xMemoryOut, xMemoryIn := "SS1_CPU1215_DI_Vars".DI11.xMemoryIn, cMemory := "SS1_CPU1215_DI_Vars".DI11.cMemory, iCounterIn := "SS1_CPU1215_DI_Vars".DI11.iCounterIn, iCounterOut := "SS1_CPU1215_DI_Vars".DI11.iCounterOut, xOutputFiltered => "SS1_CPU1215_DI_Vars".DI11.xOutput, xOutputUnFiltered => "SS1_CPU1215_DI_Vars".DI11.xInput)
   END_RUNG
   RUNG wire#powerrail
      "DIvars"(xInput := "SS1_CPU1215_DI_Vars".DI11.xOutput, iFuncSystem := "SS1_CPU1215_DI_Vars".DI11.cFuncSystemID, iFuncVar := "SS1_CPU1215_DI_Vars".DI11.cFuncVar)
   END_RUNG
   // the same network as SCL:
   "DIadv"(xInput := "DI11.01.11",
           xInversion := "SS1_CPU1215_DI_Vars".DI11.xInversion,
           cDelayOffSec := "SS1_CPU1215_DI_Vars".DI11.cDelayOffSec,
           cDelayOnSec := "SS1_CPU1215_DI_Vars".DI11.cDelayOnSec,
           xMemoryOut := "SS1_CPU1215_DI_Vars".DI11.xMemoryOut,
           xMemoryIn := "SS1_CPU1215_DI_Vars".DI11.xMemoryIn,
           cMemory := "SS1_CPU1215_DI_Vars".DI11.cMemory,
           iCounterIn := "SS1_CPU1215_DI_Vars".DI11.iCounterIn,
           iCounterOut := "SS1_CPU1215_DI_Vars".DI11.iCounterOut,
           xOutputFiltered => "SS1_CPU1215_DI_Vars".DI11.xOutput,
           xOutputUnFiltered => "SS1_CPU1215_DI_Vars".DI11.xInput);
   "DIvars"(xInput := "SS1_CPU1215_DI_Vars".DI11.xOutput,
            iFuncSystem := "SS1_CPU1215_DI_Vars".DI11.cFuncSystemID,
            iFuncVar := "SS1_CPU1215_DI_Vars".DI11.cFuncVar);
END_REGION

REGION Network 16: DIb3
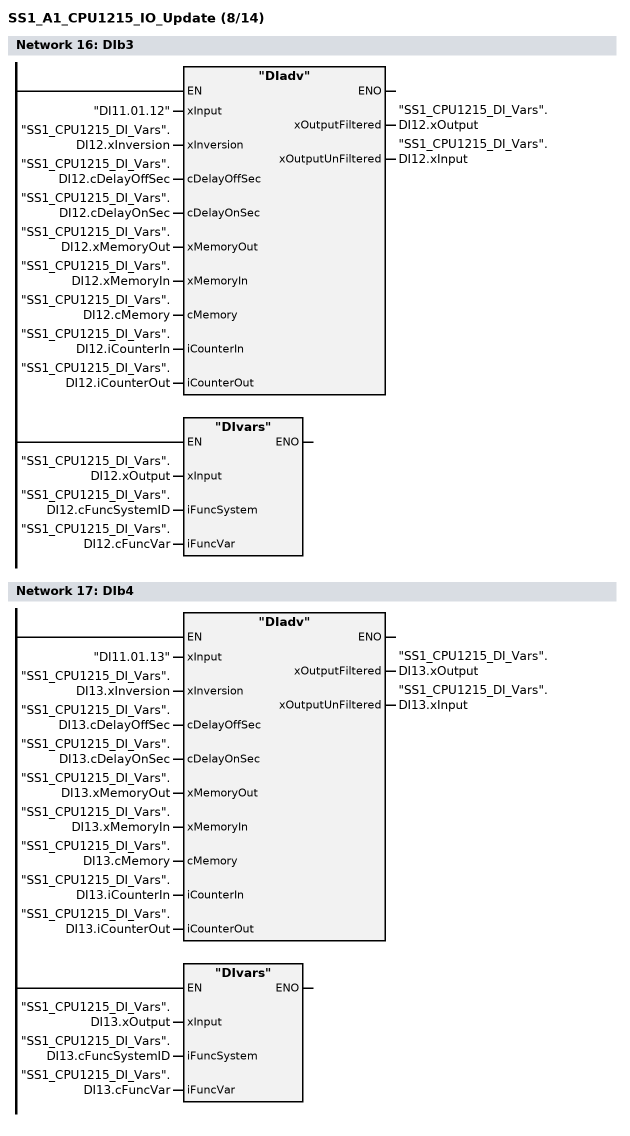
   RUNG wire#powerrail
      "DIadv"(xInput := "DI11.01.12", xInversion := "SS1_CPU1215_DI_Vars".DI12.xInversion, cDelayOffSec := "SS1_CPU1215_DI_Vars".DI12.cDelayOffSec, cDelayOnSec := "SS1_CPU1215_DI_Vars".DI12.cDelayOnSec, xMemoryOut := "SS1_CPU1215_DI_Vars".DI12.xMemoryOut, xMemoryIn := "SS1_CPU1215_DI_Vars".DI12.xMemoryIn, cMemory := "SS1_CPU1215_DI_Vars".DI12.cMemory, xOutputFiltered => "SS1_CPU1215_DI_Vars".DI12.xOutput, xOutputUnFiltered => "SS1_CPU1215_DI_Vars".DI12.xInput, iCounterIn := "SS1_CPU1215_DI_Vars".DI12.iCounterIn, iCounterOut := "SS1_CPU1215_DI_Vars".DI12.iCounterOut)
   END_RUNG
   RUNG wire#powerrail
      "DIvars"(xInput := "SS1_CPU1215_DI_Vars".DI12.xOutput, iFuncSystem := "SS1_CPU1215_DI_Vars".DI12.cFuncSystemID, iFuncVar := "SS1_CPU1215_DI_Vars".DI12.cFuncVar)
   END_RUNG
   // the same network as SCL:
   "DIadv"(xInput := "DI11.01.12",
           xInversion := "SS1_CPU1215_DI_Vars".DI12.xInversion,
           cDelayOffSec := "SS1_CPU1215_DI_Vars".DI12.cDelayOffSec,
           cDelayOnSec := "SS1_CPU1215_DI_Vars".DI12.cDelayOnSec,
           xMemoryOut := "SS1_CPU1215_DI_Vars".DI12.xMemoryOut,
           xMemoryIn := "SS1_CPU1215_DI_Vars".DI12.xMemoryIn,
           cMemory := "SS1_CPU1215_DI_Vars".DI12.cMemory,
           iCounterIn := "SS1_CPU1215_DI_Vars".DI12.iCounterIn,
           iCounterOut := "SS1_CPU1215_DI_Vars".DI12.iCounterOut,
           xOutputFiltered => "SS1_CPU1215_DI_Vars".DI12.xOutput,
           xOutputUnFiltered => "SS1_CPU1215_DI_Vars".DI12.xInput);
   "DIvars"(xInput := "SS1_CPU1215_DI_Vars".DI12.xOutput,
            iFuncSystem := "SS1_CPU1215_DI_Vars".DI12.cFuncSystemID,
            iFuncVar := "SS1_CPU1215_DI_Vars".DI12.cFuncVar);
END_REGION

REGION Network 17: DIb4
   RUNG wire#powerrail
      "DIadv"(xInput := "DI11.01.13", xInversion := "SS1_CPU1215_DI_Vars".DI13.xInversion, cDelayOffSec := "SS1_CPU1215_DI_Vars".DI13.cDelayOffSec, cDelayOnSec := "SS1_CPU1215_DI_Vars".DI13.cDelayOnSec, xMemoryOut := "SS1_CPU1215_DI_Vars".DI13.xMemoryOut, xMemoryIn := "SS1_CPU1215_DI_Vars".DI13.xMemoryIn, cMemory := "SS1_CPU1215_DI_Vars".DI13.cMemory, xOutputFiltered => "SS1_CPU1215_DI_Vars".DI13.xOutput, xOutputUnFiltered => "SS1_CPU1215_DI_Vars".DI13.xInput, iCounterIn := "SS1_CPU1215_DI_Vars".DI13.iCounterIn, iCounterOut := "SS1_CPU1215_DI_Vars".DI13.iCounterOut)
   END_RUNG
   RUNG wire#powerrail
      "DIvars"(xInput := "SS1_CPU1215_DI_Vars".DI13.xOutput, iFuncSystem := "SS1_CPU1215_DI_Vars".DI13.cFuncSystemID, iFuncVar := "SS1_CPU1215_DI_Vars".DI13.cFuncVar)
   END_RUNG
   // the same network as SCL:
   "DIadv"(xInput := "DI11.01.13",
           xInversion := "SS1_CPU1215_DI_Vars".DI13.xInversion,
           cDelayOffSec := "SS1_CPU1215_DI_Vars".DI13.cDelayOffSec,
           cDelayOnSec := "SS1_CPU1215_DI_Vars".DI13.cDelayOnSec,
           xMemoryOut := "SS1_CPU1215_DI_Vars".DI13.xMemoryOut,
           xMemoryIn := "SS1_CPU1215_DI_Vars".DI13.xMemoryIn,
           cMemory := "SS1_CPU1215_DI_Vars".DI13.cMemory,
           iCounterIn := "SS1_CPU1215_DI_Vars".DI13.iCounterIn,
           iCounterOut := "SS1_CPU1215_DI_Vars".DI13.iCounterOut,
           xOutputFiltered => "SS1_CPU1215_DI_Vars".DI13.xOutput,
           xOutputUnFiltered => "SS1_CPU1215_DI_Vars".DI13.xInput);
   "DIvars"(xInput := "SS1_CPU1215_DI_Vars".DI13.xOutput,
            iFuncSystem := "SS1_CPU1215_DI_Vars".DI13.cFuncSystemID,
            iFuncVar := "SS1_CPU1215_DI_Vars".DI13.cFuncVar);
END_REGION

REGION Network 18: DIb5 / DI01.1.14 Спрацювання охоронної сигналізації
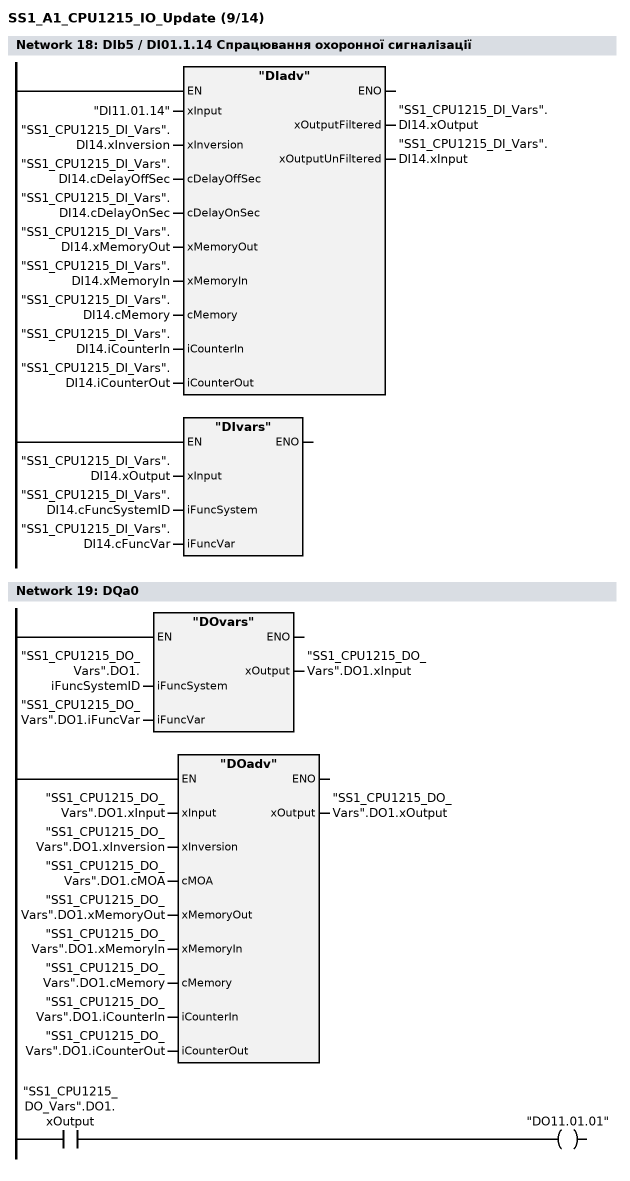
   RUNG wire#powerrail
      "DIadv"(xInput := "DI11.01.14", xInversion := "SS1_CPU1215_DI_Vars".DI14.xInversion, cDelayOffSec := "SS1_CPU1215_DI_Vars".DI14.cDelayOffSec, cDelayOnSec := "SS1_CPU1215_DI_Vars".DI14.cDelayOnSec, xMemoryOut := "SS1_CPU1215_DI_Vars".DI14.xMemoryOut, xMemoryIn := "SS1_CPU1215_DI_Vars".DI14.xMemoryIn, cMemory := "SS1_CPU1215_DI_Vars".DI14.cMemory, xOutputFiltered => "SS1_CPU1215_DI_Vars".DI14.xOutput, xOutputUnFiltered => "SS1_CPU1215_DI_Vars".DI14.xInput, iCounterIn := "SS1_CPU1215_DI_Vars".DI14.iCounterIn, iCounterOut := "SS1_CPU1215_DI_Vars".DI14.iCounterOut)
   END_RUNG
   RUNG wire#powerrail
      "DIvars"(xInput := "SS1_CPU1215_DI_Vars".DI14.xOutput, iFuncSystem := "SS1_CPU1215_DI_Vars".DI14.cFuncSystemID, iFuncVar := "SS1_CPU1215_DI_Vars".DI14.cFuncVar)
   END_RUNG
   // the same network as SCL:
   "DIadv"(xInput := "DI11.01.14",
           xInversion := "SS1_CPU1215_DI_Vars".DI14.xInversion,
           cDelayOffSec := "SS1_CPU1215_DI_Vars".DI14.cDelayOffSec,
           cDelayOnSec := "SS1_CPU1215_DI_Vars".DI14.cDelayOnSec,
           xMemoryOut := "SS1_CPU1215_DI_Vars".DI14.xMemoryOut,
           xMemoryIn := "SS1_CPU1215_DI_Vars".DI14.xMemoryIn,
           cMemory := "SS1_CPU1215_DI_Vars".DI14.cMemory,
           iCounterIn := "SS1_CPU1215_DI_Vars".DI14.iCounterIn,
           iCounterOut := "SS1_CPU1215_DI_Vars".DI14.iCounterOut,
           xOutputFiltered => "SS1_CPU1215_DI_Vars".DI14.xOutput,
           xOutputUnFiltered => "SS1_CPU1215_DI_Vars".DI14.xInput);
   "DIvars"(xInput := "SS1_CPU1215_DI_Vars".DI14.xOutput,
            iFuncSystem := "SS1_CPU1215_DI_Vars".DI14.cFuncSystemID,
            iFuncVar := "SS1_CPU1215_DI_Vars".DI14.cFuncVar);
END_REGION

REGION Network 19: DQa0
   RUNG wire#powerrail
      "DOvars"(iFuncSystem := "SS1_CPU1215_DO_Vars".DO1.iFuncSystemID, iFuncVar := "SS1_CPU1215_DO_Vars".DO1.iFuncVar, xOutput => "SS1_CPU1215_DO_Vars".DO1.xInput)
   END_RUNG
   RUNG wire#powerrail
      "DOadv"(xInput := "SS1_CPU1215_DO_Vars".DO1.xInput, xInversion := "SS1_CPU1215_DO_Vars".DO1.xInversion, cMOA := "SS1_CPU1215_DO_Vars".DO1.cMOA, xMemoryOut := "SS1_CPU1215_DO_Vars".DO1.xMemoryOut, xMemoryIn := "SS1_CPU1215_DO_Vars".DO1.xMemoryIn, cMemory := "SS1_CPU1215_DO_Vars".DO1.cMemory, xOutput => "SS1_CPU1215_DO_Vars".DO1.xOutput, iCounterIn := "SS1_CPU1215_DO_Vars".DO1.iCounterIn, iCounterOut := "SS1_CPU1215_DO_Vars".DO1.iCounterOut)
   END_RUNG
   RUNG wire#powerrail
      Contact( "SS1_CPU1215_DO_Vars".DO1.xOutput )
      Coil( "DO11.01.01" )
   END_RUNG
   // the same network as SCL:
   "DOvars"(iFuncSystem := "SS1_CPU1215_DO_Vars".DO1.iFuncSystemID,
            iFuncVar := "SS1_CPU1215_DO_Vars".DO1.iFuncVar,
            xOutput => "SS1_CPU1215_DO_Vars".DO1.xInput);
   "DOadv"(xInput := "SS1_CPU1215_DO_Vars".DO1.xInput,
           xInversion := "SS1_CPU1215_DO_Vars".DO1.xInversion,
           cMOA := "SS1_CPU1215_DO_Vars".DO1.cMOA,
           xMemoryOut := "SS1_CPU1215_DO_Vars".DO1.xMemoryOut,
           xMemoryIn := "SS1_CPU1215_DO_Vars".DO1.xMemoryIn,
           cMemory := "SS1_CPU1215_DO_Vars".DO1.cMemory,
           iCounterIn := "SS1_CPU1215_DO_Vars".DO1.iCounterIn,
           iCounterOut := "SS1_CPU1215_DO_Vars".DO1.iCounterOut,
           xOutput => "SS1_CPU1215_DO_Vars".DO1.xOutput);
   "DO11.01.01" := "SS1_CPU1215_DO_Vars".DO1.xOutput;
END_REGION

REGION Network 20: DQa1
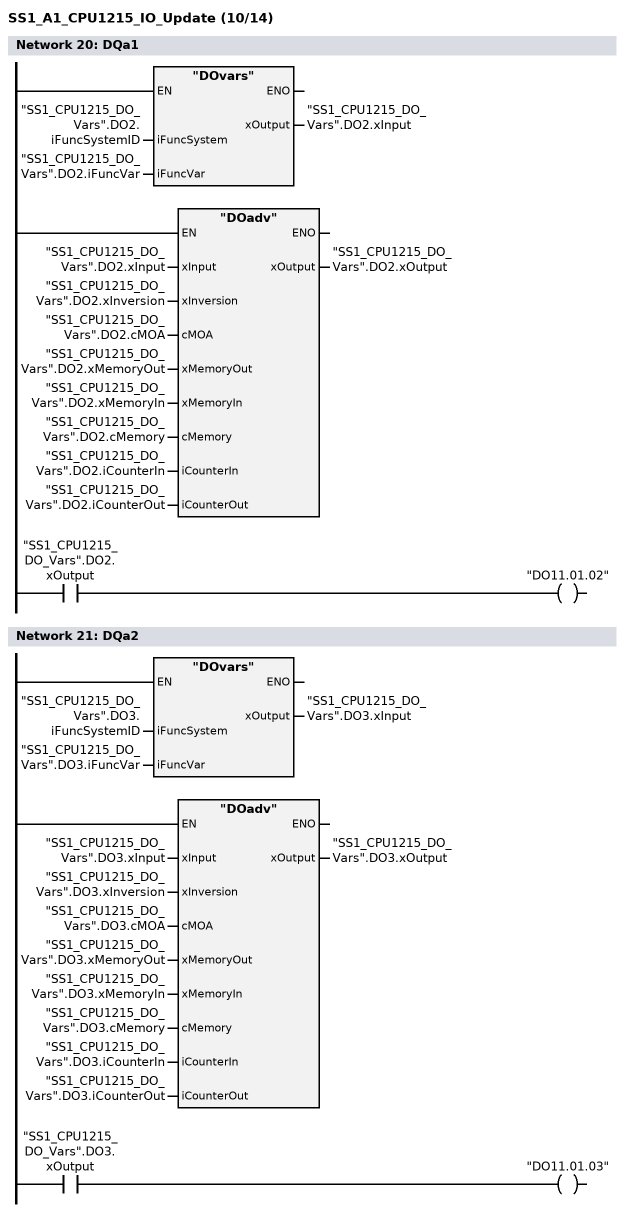
   RUNG wire#powerrail
      "DOvars"(iFuncSystem := "SS1_CPU1215_DO_Vars".DO2.iFuncSystemID, iFuncVar := "SS1_CPU1215_DO_Vars".DO2.iFuncVar, xOutput => "SS1_CPU1215_DO_Vars".DO2.xInput)
   END_RUNG
   RUNG wire#powerrail
      "DOadv"(xInput := "SS1_CPU1215_DO_Vars".DO2.xInput, xInversion := "SS1_CPU1215_DO_Vars".DO2.xInversion, cMOA := "SS1_CPU1215_DO_Vars".DO2.cMOA, xMemoryOut := "SS1_CPU1215_DO_Vars".DO2.xMemoryOut, xMemoryIn := "SS1_CPU1215_DO_Vars".DO2.xMemoryIn, cMemory := "SS1_CPU1215_DO_Vars".DO2.cMemory, xOutput => "SS1_CPU1215_DO_Vars".DO2.xOutput, iCounterIn := "SS1_CPU1215_DO_Vars".DO2.iCounterIn, iCounterOut := "SS1_CPU1215_DO_Vars".DO2.iCounterOut)
   END_RUNG
   RUNG wire#powerrail
      Contact( "SS1_CPU1215_DO_Vars".DO2.xOutput )
      Coil( "DO11.01.02" )
   END_RUNG
   // the same network as SCL:
   "DOvars"(iFuncSystem := "SS1_CPU1215_DO_Vars".DO2.iFuncSystemID,
            iFuncVar := "SS1_CPU1215_DO_Vars".DO2.iFuncVar,
            xOutput => "SS1_CPU1215_DO_Vars".DO2.xInput);
   "DOadv"(xInput := "SS1_CPU1215_DO_Vars".DO2.xInput,
           xInversion := "SS1_CPU1215_DO_Vars".DO2.xInversion,
           cMOA := "SS1_CPU1215_DO_Vars".DO2.cMOA,
           xMemoryOut := "SS1_CPU1215_DO_Vars".DO2.xMemoryOut,
           xMemoryIn := "SS1_CPU1215_DO_Vars".DO2.xMemoryIn,
           cMemory := "SS1_CPU1215_DO_Vars".DO2.cMemory,
           iCounterIn := "SS1_CPU1215_DO_Vars".DO2.iCounterIn,
           iCounterOut := "SS1_CPU1215_DO_Vars".DO2.iCounterOut,
           xOutput => "SS1_CPU1215_DO_Vars".DO2.xOutput);
   "DO11.01.02" := "SS1_CPU1215_DO_Vars".DO2.xOutput;
END_REGION

REGION Network 21: DQa2
   RUNG wire#powerrail
      "DOvars"(iFuncSystem := "SS1_CPU1215_DO_Vars".DO3.iFuncSystemID, iFuncVar := "SS1_CPU1215_DO_Vars".DO3.iFuncVar, xOutput => "SS1_CPU1215_DO_Vars".DO3.xInput)
   END_RUNG
   RUNG wire#powerrail
      "DOadv"(xInput := "SS1_CPU1215_DO_Vars".DO3.xInput, xInversion := "SS1_CPU1215_DO_Vars".DO3.xInversion, cMOA := "SS1_CPU1215_DO_Vars".DO3.cMOA, xMemoryOut := "SS1_CPU1215_DO_Vars".DO3.xMemoryOut, xMemoryIn := "SS1_CPU1215_DO_Vars".DO3.xMemoryIn, cMemory := "SS1_CPU1215_DO_Vars".DO3.cMemory, xOutput => "SS1_CPU1215_DO_Vars".DO3.xOutput, iCounterIn := "SS1_CPU1215_DO_Vars".DO3.iCounterIn, iCounterOut := "SS1_CPU1215_DO_Vars".DO3.iCounterOut)
   END_RUNG
   RUNG wire#powerrail
      Contact( "SS1_CPU1215_DO_Vars".DO3.xOutput )
      Coil( "DO11.01.03" )
   END_RUNG
   // the same network as SCL:
   "DOvars"(iFuncSystem := "SS1_CPU1215_DO_Vars".DO3.iFuncSystemID,
            iFuncVar := "SS1_CPU1215_DO_Vars".DO3.iFuncVar,
            xOutput => "SS1_CPU1215_DO_Vars".DO3.xInput);
   "DOadv"(xInput := "SS1_CPU1215_DO_Vars".DO3.xInput,
           xInversion := "SS1_CPU1215_DO_Vars".DO3.xInversion,
           cMOA := "SS1_CPU1215_DO_Vars".DO3.cMOA,
           xMemoryOut := "SS1_CPU1215_DO_Vars".DO3.xMemoryOut,
           xMemoryIn := "SS1_CPU1215_DO_Vars".DO3.xMemoryIn,
           cMemory := "SS1_CPU1215_DO_Vars".DO3.cMemory,
           iCounterIn := "SS1_CPU1215_DO_Vars".DO3.iCounterIn,
           iCounterOut := "SS1_CPU1215_DO_Vars".DO3.iCounterOut,
           xOutput => "SS1_CPU1215_DO_Vars".DO3.xOutput);
   "DO11.01.03" := "SS1_CPU1215_DO_Vars".DO3.xOutput;
END_REGION

REGION Network 22: DQa3
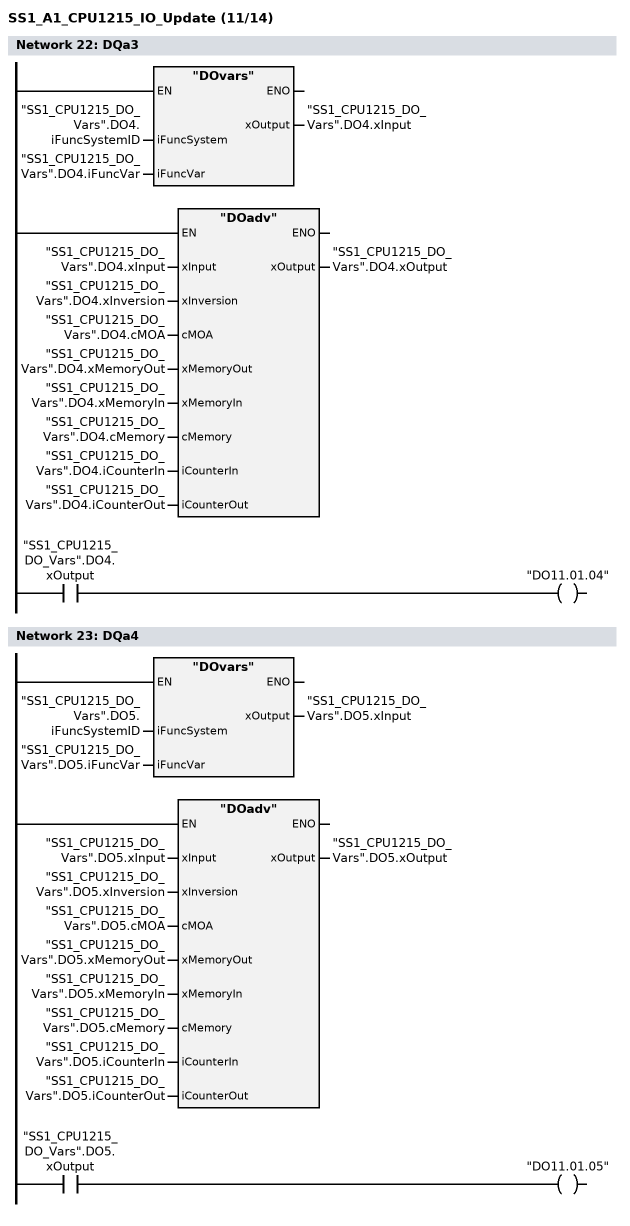
   RUNG wire#powerrail
      "DOvars"(iFuncSystem := "SS1_CPU1215_DO_Vars".DO4.iFuncSystemID, iFuncVar := "SS1_CPU1215_DO_Vars".DO4.iFuncVar, xOutput => "SS1_CPU1215_DO_Vars".DO4.xInput)
   END_RUNG
   RUNG wire#powerrail
      "DOadv"(xInput := "SS1_CPU1215_DO_Vars".DO4.xInput, xInversion := "SS1_CPU1215_DO_Vars".DO4.xInversion, cMOA := "SS1_CPU1215_DO_Vars".DO4.cMOA, xMemoryOut := "SS1_CPU1215_DO_Vars".DO4.xMemoryOut, xMemoryIn := "SS1_CPU1215_DO_Vars".DO4.xMemoryIn, cMemory := "SS1_CPU1215_DO_Vars".DO4.cMemory, xOutput => "SS1_CPU1215_DO_Vars".DO4.xOutput, iCounterIn := "SS1_CPU1215_DO_Vars".DO4.iCounterIn, iCounterOut := "SS1_CPU1215_DO_Vars".DO4.iCounterOut)
   END_RUNG
   RUNG wire#powerrail
      Contact( "SS1_CPU1215_DO_Vars".DO4.xOutput )
      Coil( "DO11.01.04" )
   END_RUNG
   // the same network as SCL:
   "DOvars"(iFuncSystem := "SS1_CPU1215_DO_Vars".DO4.iFuncSystemID,
            iFuncVar := "SS1_CPU1215_DO_Vars".DO4.iFuncVar,
            xOutput => "SS1_CPU1215_DO_Vars".DO4.xInput);
   "DOadv"(xInput := "SS1_CPU1215_DO_Vars".DO4.xInput,
           xInversion := "SS1_CPU1215_DO_Vars".DO4.xInversion,
           cMOA := "SS1_CPU1215_DO_Vars".DO4.cMOA,
           xMemoryOut := "SS1_CPU1215_DO_Vars".DO4.xMemoryOut,
           xMemoryIn := "SS1_CPU1215_DO_Vars".DO4.xMemoryIn,
           cMemory := "SS1_CPU1215_DO_Vars".DO4.cMemory,
           iCounterIn := "SS1_CPU1215_DO_Vars".DO4.iCounterIn,
           iCounterOut := "SS1_CPU1215_DO_Vars".DO4.iCounterOut,
           xOutput => "SS1_CPU1215_DO_Vars".DO4.xOutput);
   "DO11.01.04" := "SS1_CPU1215_DO_Vars".DO4.xOutput;
END_REGION

REGION Network 23: DQa4
   RUNG wire#powerrail
      "DOvars"(iFuncSystem := "SS1_CPU1215_DO_Vars".DO5.iFuncSystemID, iFuncVar := "SS1_CPU1215_DO_Vars".DO5.iFuncVar, xOutput => "SS1_CPU1215_DO_Vars".DO5.xInput)
   END_RUNG
   RUNG wire#powerrail
      "DOadv"(xInput := "SS1_CPU1215_DO_Vars".DO5.xInput, xInversion := "SS1_CPU1215_DO_Vars".DO5.xInversion, cMOA := "SS1_CPU1215_DO_Vars".DO5.cMOA, xMemoryOut := "SS1_CPU1215_DO_Vars".DO5.xMemoryOut, xMemoryIn := "SS1_CPU1215_DO_Vars".DO5.xMemoryIn, cMemory := "SS1_CPU1215_DO_Vars".DO5.cMemory, xOutput => "SS1_CPU1215_DO_Vars".DO5.xOutput, iCounterIn := "SS1_CPU1215_DO_Vars".DO5.iCounterIn, iCounterOut := "SS1_CPU1215_DO_Vars".DO5.iCounterOut)
   END_RUNG
   RUNG wire#powerrail
      Contact( "SS1_CPU1215_DO_Vars".DO5.xOutput )
      Coil( "DO11.01.05" )
   END_RUNG
   // the same network as SCL:
   "DOvars"(iFuncSystem := "SS1_CPU1215_DO_Vars".DO5.iFuncSystemID,
            iFuncVar := "SS1_CPU1215_DO_Vars".DO5.iFuncVar,
            xOutput => "SS1_CPU1215_DO_Vars".DO5.xInput);
   "DOadv"(xInput := "SS1_CPU1215_DO_Vars".DO5.xInput,
           xInversion := "SS1_CPU1215_DO_Vars".DO5.xInversion,
           cMOA := "SS1_CPU1215_DO_Vars".DO5.cMOA,
           xMemoryOut := "SS1_CPU1215_DO_Vars".DO5.xMemoryOut,
           xMemoryIn := "SS1_CPU1215_DO_Vars".DO5.xMemoryIn,
           cMemory := "SS1_CPU1215_DO_Vars".DO5.cMemory,
           iCounterIn := "SS1_CPU1215_DO_Vars".DO5.iCounterIn,
           iCounterOut := "SS1_CPU1215_DO_Vars".DO5.iCounterOut,
           xOutput => "SS1_CPU1215_DO_Vars".DO5.xOutput);
   "DO11.01.05" := "SS1_CPU1215_DO_Vars".DO5.xOutput;
END_REGION

REGION Network 24: DQa5
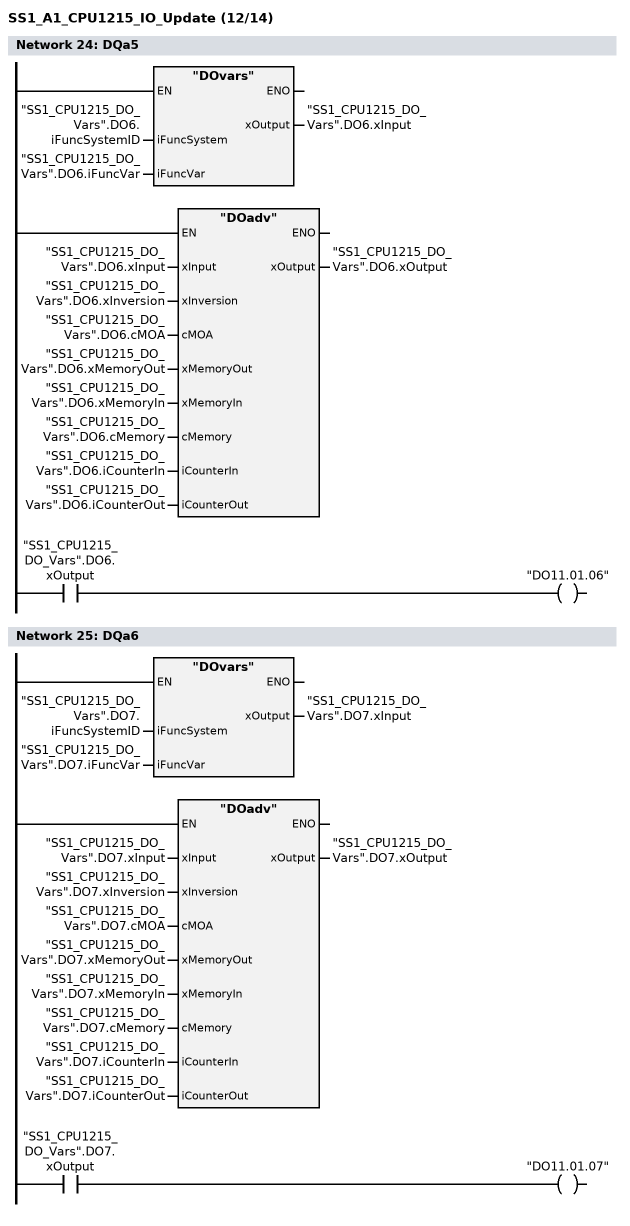
   RUNG wire#powerrail
      "DOvars"(iFuncSystem := "SS1_CPU1215_DO_Vars".DO6.iFuncSystemID, iFuncVar := "SS1_CPU1215_DO_Vars".DO6.iFuncVar, xOutput => "SS1_CPU1215_DO_Vars".DO6.xInput)
   END_RUNG
   RUNG wire#powerrail
      "DOadv"(xInput := "SS1_CPU1215_DO_Vars".DO6.xInput, xInversion := "SS1_CPU1215_DO_Vars".DO6.xInversion, cMOA := "SS1_CPU1215_DO_Vars".DO6.cMOA, xMemoryOut := "SS1_CPU1215_DO_Vars".DO6.xMemoryOut, xMemoryIn := "SS1_CPU1215_DO_Vars".DO6.xMemoryIn, cMemory := "SS1_CPU1215_DO_Vars".DO6.cMemory, xOutput => "SS1_CPU1215_DO_Vars".DO6.xOutput, iCounterIn := "SS1_CPU1215_DO_Vars".DO6.iCounterIn, iCounterOut := "SS1_CPU1215_DO_Vars".DO6.iCounterOut)
   END_RUNG
   RUNG wire#powerrail
      Contact( "SS1_CPU1215_DO_Vars".DO6.xOutput )
      Coil( "DO11.01.06" )
   END_RUNG
   // the same network as SCL:
   "DOvars"(iFuncSystem := "SS1_CPU1215_DO_Vars".DO6.iFuncSystemID,
            iFuncVar := "SS1_CPU1215_DO_Vars".DO6.iFuncVar,
            xOutput => "SS1_CPU1215_DO_Vars".DO6.xInput);
   "DOadv"(xInput := "SS1_CPU1215_DO_Vars".DO6.xInput,
           xInversion := "SS1_CPU1215_DO_Vars".DO6.xInversion,
           cMOA := "SS1_CPU1215_DO_Vars".DO6.cMOA,
           xMemoryOut := "SS1_CPU1215_DO_Vars".DO6.xMemoryOut,
           xMemoryIn := "SS1_CPU1215_DO_Vars".DO6.xMemoryIn,
           cMemory := "SS1_CPU1215_DO_Vars".DO6.cMemory,
           iCounterIn := "SS1_CPU1215_DO_Vars".DO6.iCounterIn,
           iCounterOut := "SS1_CPU1215_DO_Vars".DO6.iCounterOut,
           xOutput => "SS1_CPU1215_DO_Vars".DO6.xOutput);
   "DO11.01.06" := "SS1_CPU1215_DO_Vars".DO6.xOutput;
END_REGION

REGION Network 25: DQa6
   RUNG wire#powerrail
      "DOvars"(iFuncSystem := "SS1_CPU1215_DO_Vars".DO7.iFuncSystemID, iFuncVar := "SS1_CPU1215_DO_Vars".DO7.iFuncVar, xOutput => "SS1_CPU1215_DO_Vars".DO7.xInput)
   END_RUNG
   RUNG wire#powerrail
      "DOadv"(xInput := "SS1_CPU1215_DO_Vars".DO7.xInput, xInversion := "SS1_CPU1215_DO_Vars".DO7.xInversion, cMOA := "SS1_CPU1215_DO_Vars".DO7.cMOA, xMemoryOut := "SS1_CPU1215_DO_Vars".DO7.xMemoryOut, xMemoryIn := "SS1_CPU1215_DO_Vars".DO7.xMemoryIn, cMemory := "SS1_CPU1215_DO_Vars".DO7.cMemory, xOutput => "SS1_CPU1215_DO_Vars".DO7.xOutput, iCounterIn := "SS1_CPU1215_DO_Vars".DO7.iCounterIn, iCounterOut := "SS1_CPU1215_DO_Vars".DO7.iCounterOut)
   END_RUNG
   RUNG wire#powerrail
      Contact( "SS1_CPU1215_DO_Vars".DO7.xOutput )
      Coil( "DO11.01.07" )
   END_RUNG
   // the same network as SCL:
   "DOvars"(iFuncSystem := "SS1_CPU1215_DO_Vars".DO7.iFuncSystemID,
            iFuncVar := "SS1_CPU1215_DO_Vars".DO7.iFuncVar,
            xOutput => "SS1_CPU1215_DO_Vars".DO7.xInput);
   "DOadv"(xInput := "SS1_CPU1215_DO_Vars".DO7.xInput,
           xInversion := "SS1_CPU1215_DO_Vars".DO7.xInversion,
           cMOA := "SS1_CPU1215_DO_Vars".DO7.cMOA,
           xMemoryOut := "SS1_CPU1215_DO_Vars".DO7.xMemoryOut,
           xMemoryIn := "SS1_CPU1215_DO_Vars".DO7.xMemoryIn,
           cMemory := "SS1_CPU1215_DO_Vars".DO7.cMemory,
           iCounterIn := "SS1_CPU1215_DO_Vars".DO7.iCounterIn,
           iCounterOut := "SS1_CPU1215_DO_Vars".DO7.iCounterOut,
           xOutput => "SS1_CPU1215_DO_Vars".DO7.xOutput);
   "DO11.01.07" := "SS1_CPU1215_DO_Vars".DO7.xOutput;
END_REGION

REGION Network 26: DQa7
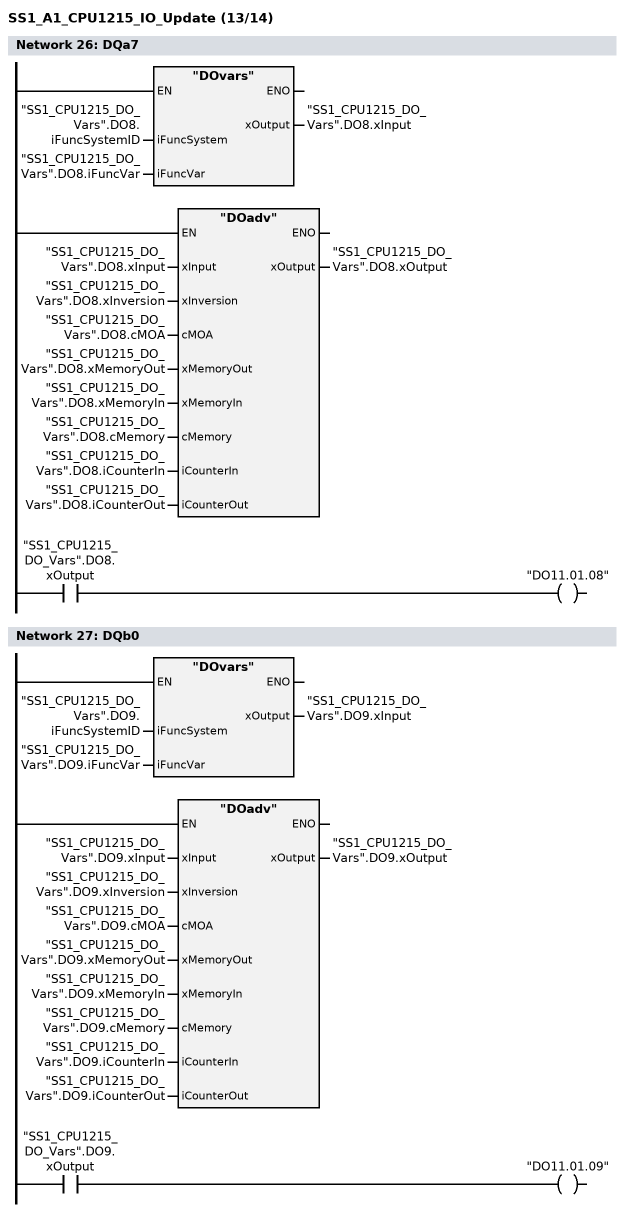
   RUNG wire#powerrail
      "DOvars"(iFuncSystem := "SS1_CPU1215_DO_Vars".DO8.iFuncSystemID, iFuncVar := "SS1_CPU1215_DO_Vars".DO8.iFuncVar, xOutput => "SS1_CPU1215_DO_Vars".DO8.xInput)
   END_RUNG
   RUNG wire#powerrail
      "DOadv"(xInput := "SS1_CPU1215_DO_Vars".DO8.xInput, xInversion := "SS1_CPU1215_DO_Vars".DO8.xInversion, cMOA := "SS1_CPU1215_DO_Vars".DO8.cMOA, xMemoryOut := "SS1_CPU1215_DO_Vars".DO8.xMemoryOut, xMemoryIn := "SS1_CPU1215_DO_Vars".DO8.xMemoryIn, cMemory := "SS1_CPU1215_DO_Vars".DO8.cMemory, xOutput => "SS1_CPU1215_DO_Vars".DO8.xOutput, iCounterIn := "SS1_CPU1215_DO_Vars".DO8.iCounterIn, iCounterOut := "SS1_CPU1215_DO_Vars".DO8.iCounterOut)
   END_RUNG
   RUNG wire#powerrail
      Contact( "SS1_CPU1215_DO_Vars".DO8.xOutput )
      Coil( "DO11.01.08" )
   END_RUNG
   // the same network as SCL:
   "DOvars"(iFuncSystem := "SS1_CPU1215_DO_Vars".DO8.iFuncSystemID,
            iFuncVar := "SS1_CPU1215_DO_Vars".DO8.iFuncVar,
            xOutput => "SS1_CPU1215_DO_Vars".DO8.xInput);
   "DOadv"(xInput := "SS1_CPU1215_DO_Vars".DO8.xInput,
           xInversion := "SS1_CPU1215_DO_Vars".DO8.xInversion,
           cMOA := "SS1_CPU1215_DO_Vars".DO8.cMOA,
           xMemoryOut := "SS1_CPU1215_DO_Vars".DO8.xMemoryOut,
           xMemoryIn := "SS1_CPU1215_DO_Vars".DO8.xMemoryIn,
           cMemory := "SS1_CPU1215_DO_Vars".DO8.cMemory,
           iCounterIn := "SS1_CPU1215_DO_Vars".DO8.iCounterIn,
           iCounterOut := "SS1_CPU1215_DO_Vars".DO8.iCounterOut,
           xOutput => "SS1_CPU1215_DO_Vars".DO8.xOutput);
   "DO11.01.08" := "SS1_CPU1215_DO_Vars".DO8.xOutput;
END_REGION

REGION Network 27: DQb0
   RUNG wire#powerrail
      "DOvars"(iFuncSystem := "SS1_CPU1215_DO_Vars".DO9.iFuncSystemID, iFuncVar := "SS1_CPU1215_DO_Vars".DO9.iFuncVar, xOutput => "SS1_CPU1215_DO_Vars".DO9.xInput)
   END_RUNG
   RUNG wire#powerrail
      "DOadv"(xInput := "SS1_CPU1215_DO_Vars".DO9.xInput, xInversion := "SS1_CPU1215_DO_Vars".DO9.xInversion, cMOA := "SS1_CPU1215_DO_Vars".DO9.cMOA, xMemoryOut := "SS1_CPU1215_DO_Vars".DO9.xMemoryOut, xMemoryIn := "SS1_CPU1215_DO_Vars".DO9.xMemoryIn, cMemory := "SS1_CPU1215_DO_Vars".DO9.cMemory, xOutput => "SS1_CPU1215_DO_Vars".DO9.xOutput, iCounterIn := "SS1_CPU1215_DO_Vars".DO9.iCounterIn, iCounterOut := "SS1_CPU1215_DO_Vars".DO9.iCounterOut)
   END_RUNG
   RUNG wire#powerrail
      Contact( "SS1_CPU1215_DO_Vars".DO9.xOutput )
      Coil( "DO11.01.09" )
   END_RUNG
   // the same network as SCL:
   "DOvars"(iFuncSystem := "SS1_CPU1215_DO_Vars".DO9.iFuncSystemID,
            iFuncVar := "SS1_CPU1215_DO_Vars".DO9.iFuncVar,
            xOutput => "SS1_CPU1215_DO_Vars".DO9.xInput);
   "DOadv"(xInput := "SS1_CPU1215_DO_Vars".DO9.xInput,
           xInversion := "SS1_CPU1215_DO_Vars".DO9.xInversion,
           cMOA := "SS1_CPU1215_DO_Vars".DO9.cMOA,
           xMemoryOut := "SS1_CPU1215_DO_Vars".DO9.xMemoryOut,
           xMemoryIn := "SS1_CPU1215_DO_Vars".DO9.xMemoryIn,
           cMemory := "SS1_CPU1215_DO_Vars".DO9.cMemory,
           iCounterIn := "SS1_CPU1215_DO_Vars".DO9.iCounterIn,
           iCounterOut := "SS1_CPU1215_DO_Vars".DO9.iCounterOut,
           xOutput => "SS1_CPU1215_DO_Vars".DO9.xOutput);
   "DO11.01.09" := "SS1_CPU1215_DO_Vars".DO9.xOutput;
END_REGION

REGION Network 28: DQb1
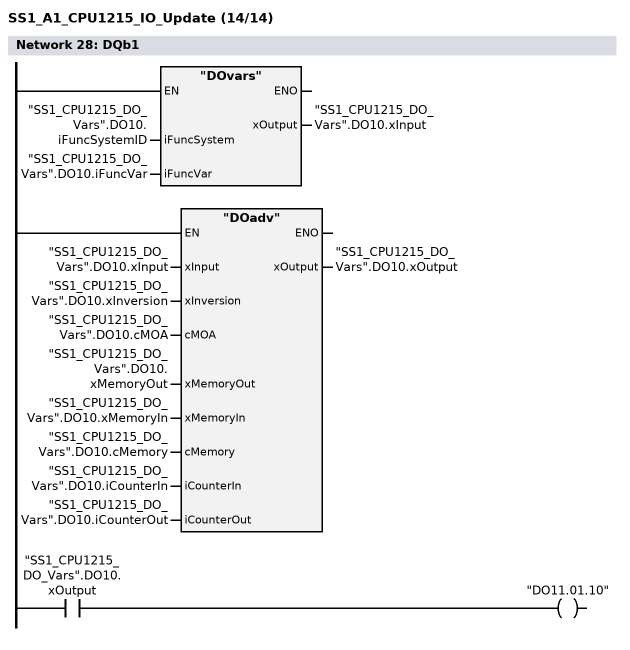
   RUNG wire#powerrail
      "DOvars"(iFuncSystem := "SS1_CPU1215_DO_Vars".DO10.iFuncSystemID, iFuncVar := "SS1_CPU1215_DO_Vars".DO10.iFuncVar, xOutput => "SS1_CPU1215_DO_Vars".DO10.xInput)
   END_RUNG
   RUNG wire#powerrail
      "DOadv"(xInput := "SS1_CPU1215_DO_Vars".DO10.xInput, xInversion := "SS1_CPU1215_DO_Vars".DO10.xInversion, cMOA := "SS1_CPU1215_DO_Vars".DO10.cMOA, xMemoryOut := "SS1_CPU1215_DO_Vars".DO10.xMemoryOut, xMemoryIn := "SS1_CPU1215_DO_Vars".DO10.xMemoryIn, cMemory := "SS1_CPU1215_DO_Vars".DO10.cMemory, xOutput => "SS1_CPU1215_DO_Vars".DO10.xOutput, iCounterIn := "SS1_CPU1215_DO_Vars".DO10.iCounterIn, iCounterOut := "SS1_CPU1215_DO_Vars".DO10.iCounterOut)
   END_RUNG
   RUNG wire#powerrail
      Contact( "SS1_CPU1215_DO_Vars".DO10.xOutput )
      Coil( "DO11.01.10" )
   END_RUNG
   // the same network as SCL:
   "DOvars"(iFuncSystem := "SS1_CPU1215_DO_Vars".DO10.iFuncSystemID,
            iFuncVar := "SS1_CPU1215_DO_Vars".DO10.iFuncVar,
            xOutput => "SS1_CPU1215_DO_Vars".DO10.xInput);
   "DOadv"(xInput := "SS1_CPU1215_DO_Vars".DO10.xInput,
           xInversion := "SS1_CPU1215_DO_Vars".DO10.xInversion,
           cMOA := "SS1_CPU1215_DO_Vars".DO10.cMOA,
           xMemoryOut := "SS1_CPU1215_DO_Vars".DO10.xMemoryOut,
           xMemoryIn := "SS1_CPU1215_DO_Vars".DO10.xMemoryIn,
           cMemory := "SS1_CPU1215_DO_Vars".DO10.cMemory,
           iCounterIn := "SS1_CPU1215_DO_Vars".DO10.iCounterIn,
           iCounterOut := "SS1_CPU1215_DO_Vars".DO10.iCounterOut,
           xOutput => "SS1_CPU1215_DO_Vars".DO10.xOutput);
   "DO11.01.10" := "SS1_CPU1215_DO_Vars".DO10.xOutput;
END_REGION
END_FUNCTION
